{attribute addProperty BoxType "EL3773-0000-0018"}
{attribute addProperty Id "U2_SamplesAT %I*ARRAY [1..10] OF INT16020"}
{attribute addProperty CRC "4020818520"}
{attribute addProperty SizeInBites "160"}
{attribute addProperty SizeInBytes "20"}
TYPE L2_Voltage_Samples_EFA8D258 :
STRUCT
	{attribute addProperty Name "U2_Samples"}
	U2_Samples AT %I* : ARRAY [1..10] OF INT;
END_STRUCT
END_TYPE

(* stored: Version 1.2.0.0, ProductVersion 3.1.4024.9
   DUT L2_Voltage_Samples_EFA8D258: Id {6d82da9f-007e-4ccc-997a-2c08f2011dbd} *)
